// TwinCAT 3 PLC project LCLSGeneral
// Title: LCLS General
// Company: SLAC
// Author: Alex Wallace
// ProjectVersion: 0.0.0
// Description: Generally useful POUs: - Logger - FB diagnostics - EtherCAT diagnostic
// ProgramVersion: 3.1.4020.2
// libraries:
//   Tc2_EtherCAT, * (Beckhoff Automation GmbH)
//   Tc2_IoFunctions, * (Beckhoff Automation GmbH)
//   Tc2_ModbusSrv, * (Beckhoff Automation GmbH)
//   Tc2_SerialCom, * (Beckhoff Automation GmbH)
//   Tc2_Standard, * (Beckhoff Automation GmbH)
//   Tc2_System, * (Beckhoff Automation GmbH)
//   Tc2_TcpIp, * (Beckhoff Automation GmbH)
//   Tc2_Utilities, * (Beckhoff Automation GmbH)
//   Tc3_EventLogger, * (Beckhoff Automation GmbH)
//   Tc3_JsonXml, * (Beckhoff Automation GmbH)
//   Tc3_Module, * (Beckhoff Automation GmbH)
// project tree:
//   Data types/Misc/ ST_System.TcDUT (not stored)
//   GVLs/ DefaultGlobals.TcGVL, Global_Variables_EtherCAT.TcGVL (not stored)
//   POUs/Logger/ FB_LogHandler.TcPOU (not stored)
//   / Task_3.TcTTO (not stored)

// ---- GVLs/DefaultGlobals.TcGVL
//These are variables every PLC project should have
VAR_GLOBAL

    stSys	:	ST_System; //Included for you
    fTimeStamp: LREAL;
END_VAR
